VISUALIZATION Page_Infeed  // 1080x660
END_VISUALIZATION

(* stored: Version 1.1.0.1, ProductVersion 3.1.4026.13
   Visu Page_Infeed: Id {d8c6c725-09e5-4e94-a239-254f43e70ae2} *)
